PROGRAM S02_LidInjecting
VAR
	//工站
	station					: REFERENCE TO FB_Station:=fbstation[2];
	//气缸
	fbHOZAdjustCyl_1	:REFERENCE TO FB_Cylinder:=fbCylinder[7];	//	上层水平调整气缸1
//	fbHOZAdjustCyl_2	:REFERENCE TO FB_Cylinder:=fbCylinder[8];	//	上层水平调整气缸2
	fbHOZAdjustCyl_3	:REFERENCE TO FB_Cylinder:=fbCylinder[9];	//	下层水平调整气缸1
//	fbHOZAdjustCyl_4	:REFERENCE TO FB_Cylinder:=fbCylinder[10];	//	下层水平调整气缸2
	fbROTCyl	:REFERENCE TO FB_Cylinder:=fbCylinder[11];	//	旋转气缸-防滴液
	//伺服
	fbXAxisMove	 :REFERENCE TO FB_Axis:=fbAxis[3];	//	注液工位X轴伺服
	fbYAxisMove	 :REFERENCE TO FB_Axis:=fbAxis[4];	//	注液工位Y轴伺服
	fbZAxisMove	 :REFERENCE TO FB_Axis:=fbAxis[5];	//	注液工位Z轴伺服
	fbStirAxis	 :REFERENCE TO FB_Axis:=fbAxis[9];	//	磁珠搅拌
	//蠕动泵
	(*直接用全局变量*)
	//称
	fbMKC204C:REFERENCE TO FB_MT_MKC:=fbMCK204w;
	//自动校准
	fbAutoCalib	:REFERENCE TO FB_AutoCal:=fbAutoCal;

	//延时
	arTonDelay :ARRAY[1..20] OF TON;
	//返回值
	UdiReturnValue :ARRAY[1..20] OF UDINT;
	//本地过程数据
	arProcessDataStation : ARRAY [1..2] OF DUT_MainlineFixture;
	i: INT;
	xNeedCalibration: BOOL;
	// 蠕动泵校准完成
	xCalibCompleted: BOOL;
	// X轴循环
	bXCounter: BYTE;
	//过程记录
	tsModuleProcess:ARRAY[1..gc_ModuleProNo] OF DUT_Process;
	xClearModuleProcessDone:BOOL;
	bClearProcessStep	:BYTE;
	// //首次循环
	_FirstCycle: ARRAY[1..10] OF BOOL;
	//深孔板到位传感器
	xSensorReached:ARRAY[1..2] OF BOOL;
END_VAR

A_Input();
Alarm();
Delay();
FlowAuto();
FlowInit();
General();
ILC();
TipAuto();
TipManual();
Z_Output();

ACTION A_Input:
//气缸

fbHOZAdjustCyl_1.xWP_Sensor	:=	IxS02HOZAdjustCyl_1WP  AND IxS02HOZAdjustCyl_2WP	;
fbHOZAdjustCyl_1.xHP_Sensor	:=	IxS02HOZAdjustCyl_1HP	 AND IxS02HOZAdjustCyl_2HP;
fbHOZAdjustCyl_3.xWP_Sensor	:=	IxS02HOZAdjustCyl_3WP	AND IxS02HOZAdjustCyl_4WP	;
fbHOZAdjustCyl_3.xHP_Sensor	:=	IxS02HOZAdjustCyl_3HP	AND IxS02HOZAdjustCyl_4HP;;
fbROTCyl.xWP_Sensor	:=	IxS02ROTCylWP	;
fbROTCyl.xHP_Sensor	:=	IxS02ROTCylHP	;

xSensorReached[1]:=IxS02Sensor1Reached	;//	注液工位¶到位传感器1
xSensorReached[2]:=IxS02Sensor2Reached	;//	注液工位¶到位传感器2
END_ACTION

ACTION Alarm:
station.adwAlarm[1].00	:=	station.xInitTimeout	;//	S02 初始化超时
//station.adwAlarm[1].01	:=	fbRudongPump[1].xError	;//	S02注液工位蠕动泵1报错
//station.adwAlarm[1].02	:=	fbRudongPump[2].xError	;//	S02注液工位蠕动泵2报错
//station.adwAlarm[1].03	:=	fbRudongPump[3].xError	;//	S02注液工位蠕动泵3报错
//station.adwAlarm[1].04	:=	fbRudongPump[4].xError	;//	S02注液工位蠕动泵4报错
//station.adwAlarm[1].05	:=	fbRudongPump[5].xError	;//	S02注液工位蠕动泵5报错
//station.adwAlarm[1].06	:=	fbRudongPump[6].xError	;//	S02注液工位蠕动泵6报错
//station.adwAlarm[1].07	:=	fbRudongPump[7].xError	;//	S02注液工位蠕动泵7报错
//station.adwAlarm[1].08	:=	fbRudongPump[8].xError	;//	S02注液工位蠕动泵8报错
//station.adwAlarm[1].09	:=	fbRudongPump[9].xError	;//	S02注液工位蠕动泵9报错
//station.adwAlarm[1].10	:=	fbRudongPump[10].xError	;//	S02注液工位蠕动泵10报错
//station.adwAlarm[1].11	:=	fbRudongPump[11].xError	;//	S02注液工位蠕动泵11报错
//station.adwAlarm[1].12	:=	fbRudongPump[12].xError	;//	S02注液工位蠕动泵12报错
station.adwAlarm[1].13	:=	fbHOZAdjustCyl_1.xHP_Off 	;//	S02上层水平调整气缸1原点未到位
station.adwAlarm[1].14	:=	fbHOZAdjustCyl_1.xWP_Off 	;//	S02上层水平调整气缸1动点未到位
station.adwAlarm[1].15	:=	fbHOZAdjustCyl_3.xHP_Off	;//	S02下层水平调整气缸1原点未到位
station.adwAlarm[1].16	:=	fbHOZAdjustCyl_3.xWP_Off	;//	S02下层水平调整气缸1动点未到位
station.adwAlarm[1].17	:=	fbROTCyl.xHP_Off	;//	S02防滴液旋转气缸原点未到位
station.adwAlarm[1].18	:=	fbROTCyl.xWP_Off	;//	S02防滴液旋转气缸动点未到位
station.adwAlarm[1].19	:=	fbXAxisMove.xError	;//	S02注液工位X轴伺服报错
station.adwAlarm[1].20	:=	fbXAxisMove.xNotPowerOn	;//	S02注液工位X轴伺服未使能
station.adwAlarm[1].21	:=	fbXAxisMove.xMoveTimeout	;//	S02注液工位X轴伺服移动超时
station.adwAlarm[1].22	:=	fbYAxisMove.xError	;//	S02注液工位Y轴伺服报错
station.adwAlarm[1].23	:=	fbYAxisMove.xNotPowerOn	;//	S02注液工位Y轴伺服未使能
station.adwAlarm[1].24	:=	fbYAxisMove.xMoveTimeout	;//	S02注液工位Y轴伺服移动超时
station.adwAlarm[1].25	:=	fbZAxisMove.xError	;//	S02注液工位Z轴伺服报错
station.adwAlarm[1].26	:=	fbZAxisMove.xNotPowerOn	;//	S02注液工位Z轴伺服未使能
station.adwAlarm[1].27	:=	fbZAxisMove.xMoveTimeout	;//	S02注液工位Z轴伺服移动超时
//station.adwAlarm[1].28	:=	fbStirAxis.xError	;//	S02注液工位搅拌旋转伺服报错
//station.adwAlarm[1].29	:=	fbStirAxis.xNotPowerOn	;//	S02注液工位搅拌旋转伺服未使能
//station.adwAlarm[1].30	:=	fbStirAxis.xMoveTimeout	;//	S02注液工位搅拌旋转伺服移动超时
station.adwAlarm[1].31	:=	fbMKC204C.xError	;//	S03注液工位称重设备报警
END_ACTION

ACTION Delay:

(*arTonDelay[01](IN:=, PT:=T#1S , Q=> , ET=> );*)//TipAuto使用
arTonDelay[02](IN:= , PT:=T#1S , Q=> , ET=> );//注液延时使用
arTonDelay[03](IN:= , PT:=T#10S , Q=> , ET=> );
arTonDelay[04](IN:= , PT:=T#0.1S , Q=> , ET=> );
arTonDelay[05](IN:= , PT:=T#0.1S , Q=> , ET=> );
arTonDelay[06](IN:= , PT:=T#0.1S , Q=> , ET=> );
arTonDelay[07](IN:= , PT:=T#0.1S , Q=> , ET=> );
arTonDelay[08](IN:= , PT:=T#0.1S , Q=> , ET=> );
arTonDelay[09](IN:= , PT:=T#0.1S , Q=> , ET=> );
arTonDelay[10](IN:= , PT:=T#0.1S , Q=> , ET=> );
END_ACTION

ACTION FlowAuto:

//-----------------------------------------初始化是否完成判断----------------------------------------------
IF NOT station.xInitDone 
THEN
 	station.iStepAuto:=0;
 	station.xDone:=FALSE;
	station.xRunningOffProhibit := FALSE ;//运行中信号Off禁止
ELSIF station.xRunning OR  (tsModuleProcess[bXCounter+1].xProcessStarted AND  NOT tsModuleProcess[bXCounter+1].xProcessCompleted)
THEN
//-----------------------------------------动作步骤--------------------------------------------------------
CASE station.iStepAuto OF	  
	0: //----Home Step，等待启动----
		IF station.xDisabled 
			AND station.xCanRun 
			AND NOT fbMachine[1].xStopped 
			AND NOT station.xSingleRunning 
		THEN
			station.xDone:=TRUE;
		END_IF
		
		IF  station.xSingleRunning 
			OR station.xCanRun 
			AND NOT station.xDone 
			AND NOT station.xDisabled 
			AND NOT fbMachine[1].xStopped
		THEN
			station.xCycleEnable:=TRUE;
			station.xDone:= FALSE;  
			station.iStepAuto:= 10;
		END_IF
    10: //复位数据 
			FOR i:=1 TO gc_ModuleProNo BY 1 DO
				MEMSET(ADR(tsModuleProcess[i]),0,SIZEOF(tsModuleProcess[i]));
			END_FOR
			station.iStepAuto:=15;
	
	15://程序分类选择
		 //进入校准程序
		 IF NOT   fbMachine[1].xTryRun THEN
					IF  station.xSingleRunning AND stCalibration.xNeedCalibration THEN
						 stCalibration.xWindowsTrigger:=TRUE;
						 station.iStepAuto:=1000;
					ELSIF  NOT  stCalibration.xNeedCalibration THEN
						station.iStepAuto:=20;
					END_IF
		ELSE
		 			station.iStepAuto:=20;
		 END_IF
	20:////Restore_after_Estop_Process1 上载数据流程
			IF  station.xSingleRunning THEN  //OR fbMachine[1].xTryRun THEN
					station.iStepAuto :=45; 
			ELSIF tsModuleProcess[1].xProcessNotStarted AND NOT  tsModuleProcess[1].xProcessStarted THEN
					station.iStepAuto :=21; (*process not started*)
			ELSIF  tsModuleProcess[1].xProcessStarted AND NOT  tsModuleProcess[1].xProcessCompleted THEN
				 station.iStepAuto :=21 ;(*process started*)
			ELSIF  tsModuleProcess[1].xProcessCompleted AND NOT tsModuleProcess[1].xQDataCompleted  THEN
					station.iStepAuto :=30  ;(*process completed*)
			ELSIF tsModuleProcess[1].xQDataCompleted THEN
					station.iStepAuto :=30;(*Qdata completed *)
			ELSE
					station.iStepAuto :=21; 
			END_IF	
	21:	
			tsModuleProcess[1].xProcessNotStarted :=TRUE;
			station.iStepAuto :=25;
	25://数据load 
		tsModuleProcess[1].xProcessStarted:=TRUE;
		MEMCPY(ADR(arProcessDataStation[1]),ADR(arMainlineFixtureData[arCurFixtureNumStation[3]]),SIZEOF(arMainlineFixtureData[arCurFixtureNumStation[3]]));
		MEMCPY(ADR(arProcessDataStation[2]),ADR(arMainlineFixtureData[arCurFixtureNumStation[4]]),SIZEOF(arMainlineFixtureData[arCurFixtureNumStation[4]]));
		tsModuleProcess[1].xProcessCompleted:=TRUE;	
		tsModuleProcess[1].xQDataCompleted:=TRUE;	
		station.iStepAuto:= 30;

	/////产品流程开始	
	30: //判断产品状态
	//	IF NOT  fbMachine[1].xTryRun THEN
			 IF ( arProcessDataStation[1].xMaterialOnOff   AND
					arProcessDataStation[2].xMaterialOnOff ) OR
			 ( xSensorReached[1] AND   xSensorReached[2])  THEN
				 station.iStepAuto:= 40;                      
			 ELSE
				 station.iStepAuto:= 998;
			 END_IF
	//	ELSE
	//	 		station.iStepAuto:= 40;
	//	END_IF
		 	
	40://写入NOK按钮
		IF   arManualNOKHmiButton[2]  AND NOT station.xSingleRunning THEN
			station.iStepAuto:=155;
			arManualNOKHmiButton[2]:=FALSE;
		ELSE
			 station.iStepAuto:=45;
		END_IF
	//////产品流程开始
	45://循环开始次数为1，总循环为2
			 bXCounter:=1;
	    station.iStepAuto:= 50;

	50:////Restore_after_Estop_Process1/2 注液流程1/2
			IF  station.xSingleRunning  OR fbMachine[1].xTryRun THEN
					station.iStepAuto :=80; 
			ELSIF tsModuleProcess[bXCounter+1].xProcessNotStarted AND NOT  tsModuleProcess[bXCounter+1].xProcessStarted THEN
					station.iStepAuto :=100; (*process not started*)
			ELSIF  tsModuleProcess[bXCounter+1].xProcessStarted AND NOT  tsModuleProcess[bXCounter+1].xProcessCompleted THEN
				 station.iStepAuto :=155 ;(*process started*)
			ELSIF  tsModuleProcess[bXCounter+1].xProcessCompleted AND NOT tsModuleProcess[bXCounter+1].xQDataCompleted  THEN
					station.iStepAuto :=150  ;(*process completed*)
			ELSIF tsModuleProcess[bXCounter+1].xQDataCompleted THEN
					station.iStepAuto :=160;(*Qdata completed *)
			ELSE
					station.iStepAuto :=80; 
			END_IF

	80://流程未开始
			 tsModuleProcess[bXCounter+1].xProcessNotStarted:=TRUE;
		 		station.iStepAuto:= 90;
	90://水平调整气缸伸出
		IF  iBoxChoose =1 THEN
			(*上层水平调整气缸*)
			fbHOZAdjustCyl_1.xAuto :=TRUE;
		//	fbHOZAdjustCyl_2.xAuto :=TRUE;
			IF  fbHOZAdjustCyl_1.xWP_Delay THEN// AND fbHOZAdjustCyl_2.xWP_Delay  THEN
					station.iStepAuto:= 100;
			END_IF
		ELSIF  iBoxChoose= 2 THEN
			(*下层水平调整气缸*)
			fbHOZAdjustCyl_3.xAuto :=TRUE;
			//fbHOZAdjustCyl_4.xAuto :=TRUE;
			IF  fbHOZAdjustCyl_3.xWP_Delay  THEN//AND fbHOZAdjustCyl_4.xWP_Delay  THEN
					station.iStepAuto:= 100;
			END_IF
		END_IF	 
	100://XY轴去注液位置1、2
			fbXAxisMove.xMoveAuto[bXCounter+1]:=TRUE;
			fbYAxisMove.xMoveAuto[bXCounter+1]:=TRUE;
			IF fbXAxisMove.xMoveInPos[bXCounter+1]  AND fbYAxisMove.xMoveInPos[bXCounter+1]  THEN
				station.iStepAuto:=110;	
			END_IF
	110:	//防滴液气缸伸出
		fbROTCyl.xAuto:=TRUE;
		IF fbROTCyl.xWP_Delay THEN
			station.iStepAuto:=120;	
		END_IF
	120://Z轴下降去注液位置
		   fbZAxisMove.xMoveAuto[2]:=TRUE;
		IF  fbZAxisMove.xMoveInPos[2] THEN
			station.iStepAuto:=125;
		END_IF
	125://屏蔽注液
			IF   axBypassSignal[2] OR fbMachine[1].xTryRun THEN
				station.iStepAuto:=145;
			ELSE
				station.iStepAuto:=130;
			END_IF
	130://开始注液
		  tsModuleProcess[bXCounter+1].xProcessStarted:=TRUE;
		 FOR i:=1 TO  11 BY 1 DO
				IF  i MOD 2 = 0  THEN
						fbRudongPump[i].stDeviceOpe.xPull_Auto[1]:=TRUE;
				ELSE	
				 		fbRudongPump[i].stDeviceOpe.xPush_Auto[1]:=TRUE;
				END_IF
		 END_FOR
		station.iStepAuto:= 140;
	140://注液结束
					arTonDelay[02](IN:=FALSE );
					 IF    fbRudongPump[1].xdone AND
								fbRudongPump[2].xDone AND
								fbRudongPump[3].xDone AND
								 fbRudongPump[4].xDone AND
									fbRudongPump[5].xDone AND
									fbRudongPump[6].xDone AND
									fbRudongPump[7].xDone AND
								 fbRudongPump[8].xDone AND
									fbRudongPump[9].xDone AND
									fbRudongPump[10].xDone AND
									fbRudongPump[11].xDone THEN
								/// fbRudongPump[12].xDone	THEN						
						 station.iStepAuto:=141;	
					 END_IF
	141://复位		
			 FOR   i:=1 TO 11 BY 1DO
							IF   fbRudongPump[i].xDone THEN
									fbRudongPump[i].xExecute:=FALSE;
							END_IF
				END_FOR
				 station.iStepAuto:=142;	
	142://延时1S
			arTonDelay[02](IN:=TRUE , PT:=T#1S , Q=> , ET=> );
			IF   arTonDelay[02].Q THEN
			 			arTonDelay[02](IN:=FALSE );
			 			 station.iStepAuto:=145;	
			END_IF
	
	145://注液完成
		tsModuleProcess[bXCounter+1].xProcessCompleted:=TRUE;
		 station.iStepAuto:=150;	
	150://写入结果
				arProcessDataStation[bXCounter].xMaterialOnOff:=TRUE;
				arProcessDataStation[bXCounter].stProduct.xlidInjecting_OK:=TRUE;
				arProcessDataStation[bXCounter].stProduct.xlidInjecting_NOK:=FALSE;	
			 tsModuleProcess[bXCounter].xQDataCompleted:=TRUE;
			 station.iStepAuto:=160;
	155://注液失败
				arProcessDataStation[bXCounter].xMaterialOnOff:=TRUE;
				arProcessDataStation[bXCounter].stProduct.xlidInjecting_OK:=FALSE;
				arProcessDataStation[bXCounter].stProduct.xlidInjecting_NOK:=TRUE;	
				station.iStepAuto:=160;
	160://Z轴上升
		  fbZAxisMove.xMoveAuto[1]:=TRUE;
		IF  fbZAxisMove.xMoveInPos[1] THEN
			station.iStepAuto:=170;
		END_IF
	170://防滴漏气缸收回
		fbROTCyl.xAuto:=FALSE;
		IF fbROTCyl.xHP_Delay THEN
			station.iStepAuto:=180;	
		END_IF
	180://循环+1
		 	bXCounter:=bXCounter +1 ;
			station.iStepAuto:=190;
	190://检查循环次数
			IF   bXCounter<=2 THEN
				station.iStepAuto:=50;
			ELSE
				station.iStepAuto:=200;
			END_IF
	200://水平调整气缸收回
			IF  iBoxChoose =1 THEN
			(*上层水平调整气缸*)
			fbHOZAdjustCyl_1.xAuto :=FALSE;
		//	fbHOZAdjustCyl_2.xAuto :=FALSE;
			IF  fbHOZAdjustCyl_1.xHP_Delay THEN  // AND fbHOZAdjustCyl_2.xHP_Delay  THEN
					station.iStepAuto:= 210;
			END_IF
		ELSIF  iBoxChoose= 2 THEN
			(*下层水平调整气缸*)
			fbHOZAdjustCyl_3.xAuto :=FALSE;
		//	fbHOZAdjustCyl_4.xAuto :=FALSE;
			IF  fbHOZAdjustCyl_3.xHP_Delay  THEN // AND fbHOZAdjustCyl_4.xHP_Delay  THEN
					station.iStepAuto:= 210;
			END_IF
		END_IF
	210:////产品流程结束	
		station.iStepAuto:= 220;
		
	220://Restore_after_Estop_Process4 数据传输 
			IF  station.xSingleRunning THEN // OR fbMachine[1].xTryRun THEN
					station.iStepAuto :=998; 
			ELSIF tsModuleProcess[4].xProcessNotStarted AND NOT  tsModuleProcess[4].xProcessStarted THEN
					station.iStepAuto :=550; (*process not started*)
			ELSIF  tsModuleProcess[4].xProcessStarted AND NOT  tsModuleProcess[4].xProcessCompleted THEN
				 station.iStepAuto :=550 ;(*process started*)
			ELSIF  tsModuleProcess[4].xProcessCompleted AND NOT tsModuleProcess[4].xQDataCompleted  THEN
					station.iStepAuto :=560  ;(*process completed*)
			ELSIF tsModuleProcess[4].xQDataCompleted THEN
					station.iStepAuto :=999;(*Qdata completed *)
			ELSE
					station.iStepAuto :=550; 
			END_IF
	550://数据unload
			tsModuleProcess[4].xProcessNotStarted :=TRUE;
			tsModuleProcess[4].xProcessStarted :=TRUE;
			MEMCPY(ADR(arMainlineFixtureData[arCurFixtureNumStation[3]]),ADR(arProcessDataStation[1]),SIZEOF(arProcessDataStation[1]));
			MEMCPY(ADR(arMainlineFixtureData[arCurFixtureNumStation[4]]),ADR(arProcessDataStation[2]),SIZEOF(arProcessDataStation[2]));
			station.iStepAuto:= 560;
		
	560:
			tsModuleProcess[4].xProcessCompleted :=TRUE;
			station.iStepAuto:= 570;
 	570://本地数据清除
			//MEMSET(ADR(arProcessDataStation[1]),0,SIZEOF(arProcessDataStation[1]));
			//MEMSET(ADR(arProcessDataStation[2]),0,SIZEOF(arProcessDataStation[2]));
			tsModuleProcess[4].xQDataCompleted:=TRUE;
			arManualNOKHmiButton[2]:=FALSE;
			station.iStepAuto:= 998;
		
	998://----Single Run Finish----
		station.iStepAuto :=999;
		IF NOT station.xSingleContinuousRun THEN
			station.xSingleRunFlag:=FALSE;
		END_IF
		station.xCycleEnable:=FALSE;	
		station.xDone:=TRUE;
		
	999://XY伺服回参考位置
			fbXAxisMove.xMoveAuto[1]:=TRUE;
			fbYAxisMove.xMoveAuto[1]:=TRUE;
			IF fbXAxisMove.xMoveInPos[1]  AND fbYAxisMove.xMoveInPos[1]  THEN
				station.iStepAuto:=0;	
			END_IF
	(****************************************蠕动泵校准程序**************************************************)
	1000://切换窗口
			stCalibration.xWindowsTrigger:=TRUE;
			station.iStepAuto:=1010;
	1010://等待人工安装好校准工装,
		 stCalibration.strCalibHmi:='Please Load  Calibration Tool and then press Start Button ';
		IF    stCalibration.xStartButtonHmi THEN
			station.iStepAuto:=1020;
		END_IF
	1020://开始循环
			stCalibration.iXCounter:=1;
			stCalibration.iYCounter:=1;
			station.iStepAuto:=1030;
	1030://计算XY轴移动目标位置
			stCalibration.strCalibHmi:='X\Y AXis move to Target Position，please Wait it';
			fbXAxisMove.rMovePosition[4]:=fbXAxisMove.rMovePosition[5]+(stCalibration.iXCounter -1);
			fbYAxisMove.rMovePosition[4]:=fbYAxisMove.rMovePosition[5]+(stCalibration.iYCounter -1);
			station.iStepAuto:=1040;
	1040://XY轴移动到位
			fbXAxisMove.xMoveAuto[4]:=TRUE;
			fbYAxisMove.xMoveAuto[4]:=TRUE;
		IF  fbXAxisMove.xMoveInPos[4]  AND fbYAxisMove.xMoveInPos[4] THEN
			station.iStepAuto:=1050;
		END_IF
	1050://Z轴去校准位置
			fbZAxisMove.xMoveAuto[3]:=TRUE;
			IF  fbZAxisMove.xMoveInPos[3] THEN
				station.iStepAuto:=1060;
			END_IF
	1060://初始化蠕动泵
			stCalibration.strCalibHmi:='All RuDongPump is initing，please Wait it';
			fbAutoCalib.stDeviceOpe.xInit_Auto:=TRUE;
			IF fbAutoCalib.xDone THEN
					station.iStepAuto:=1070;
			END_IF
	1070://选择蠕动泵控制器
			fbAutoCal.stparIn.iPumpController:=stCalibration.iYCounter;
		    station.iStepAuto:=1080;
	1080://启动自动校准程序
			stCalibration.strCalibHmi:='Auto Calibration is Running，please Wait it';
			fbAutoCalib.stDeviceOpe.xSpecificPumpHeadCal_Auto:=TRUE;
			IF  fbAutoCalib.xDone  THEN
				 fbAutoCalib.xExecute:=FALSE;
				 station.iStepAuto:=1085;
			END_IF
	1085://Z轴回参考点
			fbZAxisMove.xMoveAuto[1]:=TRUE;
			IF   fbZAxisMove.xMoveInPos[1] THEN
				 station.iStepAuto:=1090;
			END_IF
	1090://校准完成,移动到下一个位置
			stCalibration.iXCounter:=stCalibration.iXCounter +1;
			station.iStepAuto:=1100;		
	1100://判断X轴循环 
			IF    stCalibration.iXCounter>8 THEN
					 stCalibration.iYCounter:=  stCalibration.iYCounter +1;
					 stCalibration.iXCounter:=1;
					  station.iStepAuto:=1110;
			ELSE
					 station.iStepAuto:=1030;
			END_IF
			
	1110://判断Y轴循环
			IF   stCalibration.iYCounter >12 THEN
					 stCalibration.iYCounter:=1;
					 stCalibration.iXCounter:=1;
					 station.iStepAuto:=1130;
			ELSE
					station.iStepAuto:=1120;
			END_IF
	1120://等待下一组按钮按下
			stCalibration.strCalibHmi:='Wait Press Next Button HMI';
			IF stCalibration.xNextButtonHmi THEN
				station.iStepAuto:=1030;
			END_IF
			
	1130://校准完成
			stCalibration.strCalibHmi:='Calibration Completed，wait press Completed button HMI';
			IF  stCalibration.xCompletedButtonHmi THEN
					 stCalibration.xNeedCalibration:=FALSE;	
					 station.iStepAuto:=1140;
			END_IF
	1140://再按一次完成按钮关闭当前窗口
			stCalibration.strCalibHmi:='Close Current windows，wait press Completed button HMI';
			IF  stCalibration.xCompletedButtonHmi THEN
					 stCalibration.xWindowsTrigger:=FALSE;
					 station.iStepAuto:=0;
			END_IF	

	ELSE
		;	
END_CASE
END_IF
END_ACTION

ACTION FlowInit:
IF NOT station.xIniting THEN
  station.iStepInit:=0;    
ELSE
//--------------------------------------------初始化步序----------------------------------
CASE station.iStepInit OF	
 0://  
  	IF station.xIniting THEN	
  	  station.iStepInit:=10;	
  	END_IF	
10://复位数据
	FOR   i:=1 TO 12 BY 1	DO
	 	fbRudongPump[i].xExecute:=FALSE;
	END_FOR
	FOR i:=1 TO gc_ModuleProNo BY 1 DO
				MEMSET(ADR(tsModuleProcess[i]),0,SIZEOF(tsModuleProcess[i]));
	END_FOR
	station.iStepInit :=15;
15://伺服上电
  	fbXAxisMove.xPowerInit := TRUE ;
	 fbYAxisMove.xPowerInit := TRUE ;
	 fbZAxisMove.xPowerInit := TRUE ;
	IF fbXAxisMove.xPowerOn AND   fbYAxisMove.xPowerOn AND  fbZAxisMove.xPowerOn THEN 
    	station.iStepInit:=20;	
	END_IF	
20://Z轴伺服上升
		fbZAxisMove.xMoveAuto[1]:=TRUE;
		IF fbZAxisMove.xMoveInPos[1]   THEN
			station.iStepInit:=30;	
		END_IF	
30://防滴液气缸回原
	fbROTCyl.xInit:=TRUE;
	IF fbROTCyl.xHP_Delay THEN
		station.iStepInit :=50;
	END_IF
35://停止蠕动泵
		FOR i:=1 TO gc_uiRudongPump BY 1 DO
			fbRudongPump[i].stDeviceOpe.xStop_Auto:=TRUE;
		END_FOR
			station.iStepInit :=40;
40://等待蠕动泵全部停止
		FOR i:=1 TO 12 BY 1 DO
			IF  NOT  fbRudongPump[i].xDone  THEN
					EXIT;
			ELSE  
			 	fbRudongPump[i].xExecute:=FALSE;
			END_IF
			IF  i = 12 THEN
					station.iStepInit :=45;
			END_IF
		END_FOR 
45://激活配置
		FOR i:=1 TO 12 BY 1 DO
				fbRudongPump[i].xNeedConfigurePara:=TRUE;
		END_FOR
			station.iStepInit :=50;
50://XY轴回参考位
		fbXAxisMove.xMoveAuto[1]:=TRUE;
		fbYAxisMove.xMoveAuto[1]:=TRUE;
		IF fbXAxisMove.xMoveInPos[1]  AND fbYAxisMove.xMoveInPos[1]  THEN
			station.iStepInit:=90;	
		END_IF

90://水平调整气缸收回
	fbHOZAdjustCyl_1.xInit :=TRUE;
   // fbHOZAdjustCyl_2.xInit :=TRUE;
    fbHOZAdjustCyl_3.xInit :=TRUE;
   // fbHOZAdjustCyl_4.xInit :=TRUE;
	IF  fbHOZAdjustCyl_1.xHP_Delay AND 
	//	fbHOZAdjustCyl_2.xHP_Delay AND
		fbHOZAdjustCyl_3.xHP_Delay THEN
	//	fbHOZAdjustCyl_4.xHP_Delay THEN
		station.iStepInit:=100;	
	END_IF
	
100:
		station.iStepInit:=999;	
999://初始化完成	
	station.iStepInit:=0;
	station.xInitDone:=TRUE;  
END_CASE
END_IF
END_ACTION

ACTION General:
(******************清除过程记录**********************)
CASE bClearProcessStep OF
	0:	
		IF	 S08_MainLine.xClearProcessStatus THEN
			FOR i:=1 TO gc_ModuleProNo BY 1 DO
				MEMSET(ADR(tsModuleProcess[i]),0,SIZEOF(tsModuleProcess[i]));
			END_FOR
			bClearProcessStep:=10;
		END_IF
	10:
		xClearModuleProcessDone:=TRUE;
		bClearProcessStep:=20;
	20:
		IF NOT S08_MainLine.xClearProcessStatus THEN
			xClearModuleProcessDone:=FALSE;
			bClearProcessStep:=30;
		END_IF
	30:  
			bClearProcessStep:=0;
END_CASE

//测试
FOR  i:=1 TO 12 BY 1 DO
fbRudongPump[i].xNeedConfigurePara:=FALSE; 
END_FOR
END_ACTION

ACTION ILC:

//---------------------------------------------------工站可执行-------------------------------------------------------
station.xCanRun :=TRUE ;

//---------------------------------------------------气缸动作条件-------------------------------------------
fbHOZAdjustCyl_1.xOffILC	:=	TRUE	;
fbHOZAdjustCyl_1.xOnILC	:=	TRUE	;
//fbHOZAdjustCyl_2.xOffILC	:=	TRUE	;
//fbHOZAdjustCyl_2.xOnILC	:=	TRUE	;
fbHOZAdjustCyl_3.xOffILC	:=	TRUE	;
fbHOZAdjustCyl_3.xOnILC	:=	TRUE	;
//fbHOZAdjustCyl_4.xOffILC	:=	TRUE	;
//fbHOZAdjustCyl_4.xOnILC	:=	TRUE	;
fbROTCyl.xOffILC	:=	TRUE	;
fbROTCyl.xOnILC	:=	TRUE;

//---------------------------------------------------伺服动作条件-------------------------------------------
fbXAxisMove.xRunILC := 					
fbXAxisMove.xMoveILC[1] :=					
fbxAxisMove.xMoveILC[2] :=					
fbxAxisMove.xMoveILC[3] :=					
fbxAxisMove.xMoveILC[4] :=					
fbxAxisMove.xMoveILC[5] := 	TRUE;//	fbZAxisMove.xMoveInPos[1] 			;
fbYAxisMove.xRunILC := 					
fbYAxisMove.xMoveILC[1] :=					
fbYAxisMove.xMoveILC[2] :=					
fbYAxisMove.xMoveILC[3] :=					
fbYAxisMove.xMoveILC[4] :=					
fbYAxisMove.xMoveILC[5] := TRUE;//		fbZAxisMove.xMoveInPos[1] 			;
fbZAxisMove.xRunILC := 	 				
fbZAxisMove.xMoveILC[1] :=					
fbZAxisMove.xMoveILC[2] :=					
fbZAxisMove.xMoveILC[3] :=					
fbZAxisMove.xMoveILC[4] :=					
fbZAxisMove.xMoveILC[5] := 		fbROTCyl.xWP_Sensor		;
fbStirAxis.xRunILC := 					
fbStirAxis.xMoveILC[1] :=					
fbStirAxis.xMoveILC[2] :=					
fbStirAxis.xMoveILC[3] :=					
fbStirAxis.xMoveILC[4] :=					
fbStirAxis.xMoveILC[5] := 		TRUE			;
///蠕动泵
fbRudongPump[1].xDeviceRunning:=
fbRudongPump[2].xDeviceRunning:=
fbRudongPump[3].xDeviceRunning:=
fbRudongPump[4].xDeviceRunning:=
fbRudongPump[5].xDeviceRunning:=
fbRudongPump[6].xDeviceRunning:=
fbRudongPump[7].xDeviceRunning:=
fbRudongPump[8].xDeviceRunning:=
fbRudongPump[9].xDeviceRunning:=
fbRudongPump[10].xDeviceRunning:=
fbRudongPump[11].xDeviceRunning:=
fbRudongPump[12].xDeviceRunning:=station.xSingleRunning OR station.xRunning OR station.xIniting;
//称
fbMKC204C.xDeviceRunning:=station.xSingleRunning OR station.xRunning OR station.xIniting;;
END_ACTION

ACTION TipAuto:

//------------------------------------------------AutoTip Cylinder--------------------------------
station.adwAutoTip[1].00	:=	fbHOZAdjustCyl_1.xAutoTip	;
//station.adwAutoTip[1].01	:=	fbHOZAdjustCyl_2.xAutoTip	;
station.adwAutoTip[1].02	:=	fbHOZAdjustCyl_3.xAutoTip	;
//station.adwAutoTip[1].03	:=	fbHOZAdjustCyl_4.xAutoTip	;
station.adwAutoTip[1].04	:=	fbROTCyl.xAutoTip	;

//------------------------------------------------AutoTip Servo--------------------------------
//**************************************
FOR i:= 1 TO 5 BY 1 DO 
	IF fbXAxisMove.xMoveAuto[i] THEN
		fbXAxisMove.iPosNumber := i ;
	END_IF
	IF fbYAxisMove.xMoveAuto[i] THEN
		fbYAxisMove.iPosNumber := i ;
	END_IF
	IF fbZAxisMove.xMoveAuto[i] THEN
		fbZAxisMove.iPosNumber := i ;
	END_IF
	IF fbStirAxis.xMoveAuto[i] THEN
		fbStirAxis.iPosNumber := i ;
	END_IF
END_FOR


IF  fbMachine[1].xAutoMode AND NOT fbMachine[1].xRunning  THEN
	  arTonDelay[01](IN:=True , PT:=T#1S , Q=> , ET=> );
else
	  arTonDelay[01](IN:=false);
END_IF
IF arTonDelay[1].Q  THEN 
		IF fbXAxisMove.iPosNumber=1 AND NOT fbXAxisMove.xMoveInPos[1] THEN station.adwAutoTip[1].10:=TRUE; END_IF//轴伺服自动时位置不在位置1	
		IF fbXAxisMove.iPosNumber=2 AND NOT fbXAxisMove.xMoveInPos[2] THEN station.adwAutoTip[1].11:=TRUE; END_IF//轴伺服自动时位置不在位置2	
		IF fbXAxisMove.iPosNumber=3 AND NOT fbXAxisMove.xMoveInPos[3] THEN station.adwAutoTip[1].12:=TRUE; END_IF//轴伺服自动时位置不在位置3	
		IF fbXAxisMove.iPosNumber=4 AND NOT fbXAxisMove.xMoveInPos[4] THEN station.adwAutoTip[1].13:=TRUE; END_IF//轴伺服自动时位置不在位置4	
		IF fbXAxisMove.iPosNumber=5 AND NOT fbXAxisMove.xMoveInPos[5] THEN station.adwAutoTip[1].14:=TRUE; END_IF//轴伺服自动时位置不在位置5	
		
		
		IF fbYAxisMove.iPosNumber=1 AND NOT fbYAxisMove.xMoveInPos[1] THEN station.adwAutoTip[1].15:=TRUE; END_IF//轴伺服自动时位置不在位置1	
		IF fbYAxisMove.iPosNumber=2 AND NOT fbYAxisMove.xMoveInPos[2] THEN station.adwAutoTip[1].16:=TRUE; END_IF//轴伺服自动时位置不在位置2	
		IF fbYAxisMove.iPosNumber=3 AND NOT fbYAxisMove.xMoveInPos[3] THEN station.adwAutoTip[1].17:=TRUE; END_IF//轴伺服自动时位置不在位置3	
		IF fbYAxisMove.iPosNumber=4 AND NOT fbYAxisMove.xMoveInPos[4] THEN station.adwAutoTip[1].18:=TRUE; END_IF//轴伺服自动时位置不在位置4	
		IF fbYAxisMove.iPosNumber=5 AND NOT fbYAxisMove.xMoveInPos[5] THEN station.adwAutoTip[1].19:=TRUE; END_IF//轴伺服自动时位置不在位置5	
		
		IF fbZAxisMove.iPosNumber=1 AND NOT fbZAxisMove.xMoveInPos[1] THEN station.adwAutoTip[1].20:=TRUE; END_IF//轴伺服自动时位置不在位置1	
		IF fbZAxisMove.iPosNumber=2 AND NOT fbZAxisMove.xMoveInPos[2] THEN station.adwAutoTip[1].21:=TRUE; END_IF//轴伺服自动时位置不在位置2	
		IF fbZAxisMove.iPosNumber=3 AND NOT fbZAxisMove.xMoveInPos[3] THEN station.adwAutoTip[1].22:=TRUE; END_IF//轴伺服自动时位置不在位置3	
		IF fbZAxisMove.iPosNumber=4 AND NOT fbZAxisMove.xMoveInPos[4] THEN station.adwAutoTip[1].23:=TRUE; END_IF//轴伺服自动时位置不在位置4	
		IF fbZAxisMove.iPosNumber=5 AND NOT fbZAxisMove.xMoveInPos[5] THEN station.adwAutoTip[1].24:=TRUE; END_IF//轴伺服自动时位置不在位置5	
		
		IF fbStirAxis.iPosNumber=1 AND NOT fbStirAxis.xMoveInPos[1] THEN station.adwAutoTip[1].25:=TRUE; END_IF//轴伺服自动时位置不在位置1	
		IF fbStirAxis.iPosNumber=2 AND NOT fbStirAxis.xMoveInPos[2] THEN station.adwAutoTip[1].26:=TRUE; END_IF//轴伺服自动时位置不在位置2	
		IF fbStirAxis.iPosNumber=3 AND NOT fbStirAxis.xMoveInPos[3] THEN station.adwAutoTip[1].27:=TRUE; END_IF//轴伺服自动时位置不在位置3	
		IF fbStirAxis.iPosNumber=4 AND NOT fbStirAxis.xMoveInPos[4] THEN station.adwAutoTip[1].28:=TRUE; END_IF//轴伺服自动时位置不在位置4	
		IF fbStirAxis.iPosNumber=5 AND NOT fbStirAxis.xMoveInPos[5] THEN station.adwAutoTip[1].29:=TRUE; END_IF//轴伺服自动时位置不在位置5
		
END_IF
END_ACTION

ACTION TipManual:
//--------------------------------------------ManualTip------------------------------------------------------

//-------------------------------------------气缸提示---------------------------------------------------------




/////////////////////////////////////////////////////////////////////////////////////////////////////////////////
END_ACTION

ACTION Z_Output:
(**************************气缸输出********************************)
QxS02HOZAdjustCyl_1WP	:=	fbHOZAdjustCyl_1.xWP_Valve	;
QxS02HOZAdjustCyl_1HP	:=	fbHOZAdjustCyl_1.xHP_Valve	;

QxS02HOZAdjustCyl_3WP	:=	fbHOZAdjustCyl_3.xWP_Valve	;
QxS02HOZAdjustCyl_3HP	:=	fbHOZAdjustCyl_3.xHP_Valve	;

QxS02ROTCylWP	:=	fbROTCyl.xWP_Valve	;
QxS02ROTCylHP	:=	fbROTCyl.xHP_Valve	;
END_ACTION

END_PROGRAM

(* stored: Version 1.1.0.1, ProductVersion 3.1.4024.9
   POU S02_LidInjecting: Id {a38d9a95-fec8-438d-a2d4-6ac0d9bd8547}, SpecialFunc None
   Action A_Input: Id {36d6adff-dfed-4462-bb55-6ba3884a334f}
   Action Alarm: Id {830c4921-b54b-4c6d-a396-f5d5eb2c5278}
   Action Delay: Id {7f460a8e-34d3-43b7-a3e6-d254bf0f5a76}
   Action FlowAuto: Id {fc69cc4e-5f82-426b-8c9c-24d79ab9c947}
   Action FlowInit: Id {8e4e72d8-baa5-44fc-93c0-6a9330383516}
   Action General: Id {d03e3148-1994-42d2-bdc9-63de34bf4faa}
   Action ILC: Id {ee8acce8-8d32-4f66-8513-5ca456ae67c2}
   Action TipAuto: Id {889933b8-f42f-422c-ac8e-18312c628f99}
   Action TipManual: Id {dcbe8fa1-97b5-4dc0-a15a-a5576c2c36db}
   Action Z_Output: Id {a920c98e-67e5-48bd-a759-64030f6fb917} *)
